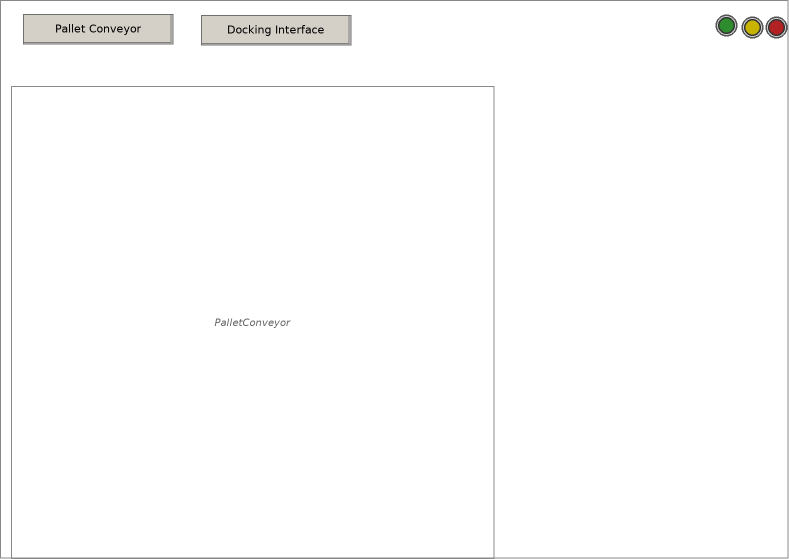
VISUALIZATION MainScreen  // 789x559
    Button (23,14 150x30), "Pallet Conveyor"
        OnMouseClick: FrameSelectionChange Selection=Selection=-1, GlobSel=AssignType=Directly, SelType=Locally
    Button (201,15 150x30), "Docking Interface"
        OnMouseClick: FrameSelectionChange Selection=Selection=-1, GlobSel=AssignType=Directly, SelType=Locally
    Frame (11,86 483x473)
        shows PalletConveyor()
        shows DockingStation()
    Lamp1 (714,13 25x25), variable: GVL_Modules.g_emUtilities.s_fbHmiLedBeaconGreen.i_bStaLed, style: Lamp-Lamp1-Green
    Lamp1 (740,15 25x25), variable: GVL_Modules.g_emUtilities.s_fbHmiLedBeaconYellow.i_bStaLed, style: Lamp-Lamp1-Yellow
    Lamp1 (764,15 25x25), variable: GVL_Modules.g_emUtilities.s_fbHmiLedBeaconRed.i_bStaLed, style: Lamp-Lamp1-Red
END_VISUALIZATION

(* stored: Version 1.1.0.1, ProductVersion 3.1.4024.12
   Visu MainScreen: Id {734abc93-732b-4b6d-9fef-18fccb00fba9} *)
